VAR_GLOBAL
	g_xFirstPass: BOOL := TRUE;
END_VAR

(* stored: Version 1.1.0.1, ProductVersion 3.1.4024.12
   GVL GVL_SAMPLE: Id {b2864d8f-27b9-49d7-a36f-f3e6d25b7296} *)
